{attribute 'enable_dynamic_creation'}
FUNCTION_BLOCK FB_Star IMPLEMENTS I_Shape
VAR_INPUT
END_VAR
VAR_OUTPUT
END_VAR
VAR
END_VAR

{warning 'Agregar implementación de método'}
METHOD M_Draw : BOOL
ADSLOGSTR(ADSLOG_MSGTYPE_HINT, 'Draw Star', '');
M_Draw := TRUE;
END_METHOD

END_FUNCTION_BLOCK

(* stored: Version 1.1.0.1, ProductVersion 3.1.4024.12
   POU FB_Star: Id {4d616224-ec60-425f-8046-aa3392519073}, SpecialFunc None
   Method M_Draw: Id {db068f4e-e9bb-4385-ae03-c5b17c4dfd7f} *)
